TYPE StateMachine :
STRUCT
	AxisGroupState : SystemState;
	SpindleState : SystemState;
END_STRUCT
END_TYPE

(* stored: Version 1.1.0.1
   DUT StateMachine: Id {8ccc48ca-66a8-486a-83a1-492780320d5a} *)
